// TwinCAT 3 PLC project PLC_Base
// ProgramVersion: 3.1.4024.0
// libraries:
//   Tc2_Standard, * (Beckhoff Automation GmbH)
//   Tc2_System, * (Beckhoff Automation GmbH)
//   Tc2_Utilities, * (Beckhoff Automation GmbH)
//   Tc3_Module, * (Beckhoff Automation GmbH)
// project tree:
//   DateAndTime/ FB_DateAndTimeHandling.TcPOU
//   EventLogging/ FB_EventLogger.TcPOU, FUN_EventTrigger.TcPOU
//   / MAIN.TcPOU, PlcTask.TcTTO
//   PersistantData/ PersistantDataHandling.TcPOU
//   PID/ FB_PI_Regulator.TcPOU, PRG_PI_Regulator_ProgramExample.TcPOU
//   Sequence Control/ FB_SequenceControl.TcPOU
// real-time tasks:
//   TASK PlcTask: cycle T#10ms, priority 20, ADS port 350
//   TASK PlcTask1: cycle T#10ms, priority 21, ADS port 351
//   TASK PlcTask2: cycle T#10ms, priority 22, ADS port 352
//   TASK PlcTask3: cycle T#10ms, priority 23, ADS port 353
// I/O:
//   DEVICE EtherCAT Master (Beckhoff), AmsNetId 10.75.2.8.2.1
//     EtherCAT Bus Coupler (EK1100) [EK1100 EtherCAT Coupler (2A E-Bus)]
//       ELM_Drive (ELM7211-9018) [ELM7211-9018 1Ch. Servo Terminal (48 V, 4,5 A RMS, OCT, STO, Safe Motion, TwinSAFE Logic)]
//         modules: Module 1 (SAFETY)
//       SafetyMaster 1 (EL1918) [EL1918, 8Ch. Safety Input 24V, TwinSAFE]
//         modules: Module 2 (FSLOGIC)
//       SafetyMaster 2 (EL1918) [EL1918, 8Ch. Safety Input 24V, TwinSAFE]
//         modules: Module 2 (FSLOGIC)
//     AX5000 (AX5206-0000-0215) [AX5206-0000-0215 EtherCAT Drive (SoE, 2 Ch.)]
//     AX8000(AX8620-0000-0105) [AX8620-0000-0105]
//       AX8000 Axis (AX8128-0220-0107) [AX8128-0220-0107 (1Ch. 28A servo axis, safe-motion, multi-FB) {v01.07_20240826.1_main_0107_AX8000_Axis_Daily}]
//         modules: Device, Device, Device, Device, Device, Device, Device, Device, Device, Device, Device (Safety), Device, Device, Device, Device, Device, Device, Device, Device, Device, Device, Device, Device, Device, Device, Device, Device, Device, Device, Device, Device, Ch A, Ch A, Ch A, Ch A, Ch A, Ch A, Ch A, Ch A, Ch A, Ch A, Ch A, Ch A, Ch A, Ch A, Ch A, Ch A, Ch A, Ch A, Ch A, Ch A, Ch A, Ch A, Ch A, Ch A, Ch A
//   DEVICE EtherCAT Master (NORDGear), AmsNetId 30.11.11.164.3.1
//     EtherCAT Slave To Insert In IO (NORDACpro) [NORDACpro]
//       modules: Module 1 (SK550P)
//   DEVICE Profinet Master (Siemens), AmsNetId 30.11.11.164.4.1
//     sinamics-g120c-pn [Siemens AG IO device SINAMICS G120C PN V4.7 with PROFINET-IO interface (RT, IRT and non-cyclic communications, PROFIsafe, Shared Device) 6SL3 210-1KExx-xxFx]
//       modules: Term 1 (DAP Module), Term 2 (Drive)
// variable links:
//   PLC_NORDGear/PLC_NORDGear Instance <-> EtherCAT Master (NORDGear)/EtherCAT Slave To Insert In IO (NORDACpro)
//     PlcTask Inputs/PRG_550P_ProgramExample.FRQ.HWin_ActualValue <-> Module 1 (SK550P)/Process data in/Actual value 1
//     PlcTask Inputs/PRG_550P_ProgramExample.FRQ.HWin_ActualValue @bit {16..64 step 16} <-> Module 1 (SK550P)/Process data in/Actual value {2..5}  (4 links)
//     PlcTask Inputs/PRG_550P_ProgramExample.FRQ.HWin_StatusWord <-> Module 1 (SK550P)/Process data in/Status word
//     PlcTask Outputs/PRG_550P_ProgramExample.FRQ.HWout_SetValue <-> Module 1 (SK550P)/Process data out/Set Value 1
//     PlcTask Outputs/PRG_550P_ProgramExample.FRQ.HWout_SetValue @bit {16..64 step 16} <-> Module 1 (SK550P)/Process data out/Set Value {2..5}  (4 links)
//     PlcTask Outputs/PRG_550P_ProgramExample.FRQ.HWout_StatusWord <-> Module 1 (SK550P)/Process data out/Control Word
//   PLC_Siemens/PLC_Siemens Instance <-> Profinet Master (Siemens)/sinamics-g120c-pn
//     PlcTask Inputs/PRG_G120C_ProgramExample.FRQ.HWin_Word <-> API/Term 2 (Drive)/Subterm 6 (Free telegram, PZD-6/6)/Inputs/Status word or actual value[0]
//     PlcTask Inputs/PRG_G120C_ProgramExample.FRQ.HWin_Word @bit {16..80 step 16} <-> API/Term 2 (Drive)/Subterm 6 (Free telegram, PZD-6/6)/Inputs/Status word or actual value[{1..5}]  (5 links)
//     PlcTask Outputs/PRG_G120C_ProgramExample.FRQ.Hwout_Word <-> API/Term 2 (Drive)/Subterm 6 (Free telegram, PZD-6/6)/Outputs/Control word or setpoint[0]
//     PlcTask Outputs/PRG_G120C_ProgramExample.FRQ.Hwout_Word @bit 16 <-> API/Term 2 (Drive)/Subterm 6 (Free telegram, PZD-6/6)/Outputs/Control word or setpoint[1]
//     PlcTask Outputs/PRG_G120C_ProgramExample.FRQ.Hwout_Word @bit 32 <-> API/Term 2 (Drive)/Subterm 6 (Free telegram, PZD-6/6)/Outputs/Control word or setpoint[2]
//     PlcTask Outputs/PRG_G120C_ProgramExample.FRQ.Hwout_Word @bit 48 <-> API/Term 2 (Drive)/Subterm 6 (Free telegram, PZD-6/6)/Outputs/Control word or setpoint[3]

CONFIGURATION PLC_Base
    RESOURCE PLC ON TwinCAT3
        TASK PlcTask(INTERVAL := T#10ms, PRIORITY := 23);
        PROGRAM MAIN WITH PlcTask : MAIN;
    END_RESOURCE
END_CONFIGURATION

// ---- MAIN.TcPOU
PROGRAM MAIN
VAR
END_VAR

PRG_PI_Regulator_ProgramExample();

END_PROGRAM

// ---- PID/PRG_PI_Regulator_ProgramExample.TcPOU
PROGRAM PRG_PI_Regulator_ProgramExample
VAR
	PID_Instance :				FB_PI_Regulator;
	Out_Error :					LREAL;
	Out_LoopOutput :			LREAL;
	Out_DutyOutput :			BOOL;
	Sts_DeadBandActive :		BOOL;
	Sts_LastReactionTime :		DINT;
	Sts_LastReactionTime_Offset :		DINT;
	SP_Old :					LREAL;
	SP_ChangeTON :				TON;
	Step_SIM :					INT;
	Step_SIM_Old :					INT;
	StepTON :					TON;
	SIMDampingFactor :			LREAL :=1.0;
	SIM_OvershootSUB :			LREAL :=10.0; 
	
END_VAR

SP_ChangeTON(IN:=PID_Instance.In_SP = SP_Old , PT:=T#2S , Q=> , ET=> );
IF SP_Old <> PID_Instance.In_SP THEN
		SP_Old := PID_Instance.In_SP;
END_IF
// PID Regulator
PID_Instance(Out_Error=>Out_Error , 
	Out_LoopOutput=>Out_LoopOutput , 
	Out_DutyOutput=>Out_DutyOutput,
	Sts_DeadBandActive=>Sts_DeadBandActive ,	
    Sts_LastReactionTime=>Sts_LastReactionTime_Offset);
	
Sts_LastReactionTime := Sts_LastReactionTime_Offset - 2000;
	
// SIM Control
	StepTON(IN:=Step_SIM_Old = Step_SIM , PT:=T#16D , Q=> , ET=> );
	IF Step_SIM_Old <> Step_SIM THEN
		Step_SIM_Old := Step_SIM;
	END_IF
	
	CASE Step_SIM OF
		
		0:
			IF StepTON.ET > INT_TO_TIME(PID_Instance.In_DutyCycle) AND SP_ChangeTON.Q THEN
				PID_Instance.In_PV := PID_Instance.In_PV + ((Out_LoopOutput) * SIMDampingFactor);	
				
				Step_SIM := 10;
			END_IF
		10:
			IF StepTON.ET > T#20MS THEN
				Step_SIM := 0;
			END_IF
			
	
	
	END_CASE

END_PROGRAM

// ---- PID/FB_PI_Regulator.TcPOU
FUNCTION_BLOCK FB_PI_Regulator
VAR_INPUT
	In_SP :				LREAL;
	In_PV :				LREAL;	
	In_DutyCycle :		INT;
	Cfg_P_Gain :		LREAL;
	Cfg_I_Gain :		LREAL;
	Cfg_D_Gain :		LREAL;
	Cfg_DeadBand :		LREAL;
	Cfg_FeedForward :	LREAL;
END_VAR
VAR_OUTPUT
	Out_Error :		LREAL;
	Out_LoopOutput :	LREAL;
	Out_DutyOutput :	BOOL;
	Sts_DeadBandActive :	BOOL;
	Sts_LastReactionTime :	DINT;
END_VAR
VAR
	
	DutyCycleTON :		TON;	
	P_LoopOutput :	LREAL;
	I_LoopOutput :	LREAL;
	
	DeadbandMin :	LREAL;
	DeadbandMax :	LREAL;
	ReactionTimeTON :	TON;
	ReactionTimeONS :	R_TRIG;
	
	Lo_DeadBandActive :	BOOL;
END_VAR

DutyCycleTON(IN:=NOT DutyCycleTON.Q , PT:=INT_TO_TIME(In_DutyCycle) , Q=> , ET=> );

// DeadBand
IF Cfg_DeadBand<> 0 THEN

IF In_PV < DeadbandMax AND In_PV > DeadbandMin THEN
	Sts_DeadBandActive :=1;
	ELSE
	Sts_DeadBandActive :=0;
END_IF

ReactionTimeONS(CLK:=Sts_DeadBandActive , Q=> );

IF ReactionTimeONS.Q THEN
	Sts_LastReactionTime := TIME_TO_DINT(ReactionTimeTON.ET);
END_IF

ReactionTimeTON(IN:= NOT Sts_DeadBandActive , PT:=T#16D , Q=> , ET=> );
ELSE
	
DeadbandMin := In_SP - 0.1;
DeadbandMax := In_SP + 0.1;	
IF In_PV < DeadbandMax AND In_PV > DeadbandMin THEN
	Lo_DeadBandActive :=1;
	ELSE
	Lo_DeadBandActive :=0;
END_IF

ReactionTimeONS(CLK:=Lo_DeadBandActive , Q=> );

IF ReactionTimeONS.Q THEN
	Sts_LastReactionTime := TIME_TO_DINT(ReactionTimeTON.ET);
END_IF

ReactionTimeTON(IN:= NOT Lo_DeadBandActive , PT:=T#16D , Q=> , ET=> );
END_IF	



//Regulation
IF DutyCycleTON.Q AND NOT Sts_DeadBandActive THEN

Out_Error := In_SP - In_PV;

// P
P_LoopOutput := Cfg_P_Gain*Out_Error;

// I
I_LoopOutput := Out_Error * Cfg_I_Gain;


// Calculate Output

Out_LoopOutput := P_LoopOutput + I_LoopOutput + Cfg_FeedForward;

END_IF

END_FUNCTION_BLOCK

// ---- DateAndTime/FB_DateAndTimeHandling.TcPOU
FUNCTION_BLOCK FB_DateAndTimeHandling
VAR_INPUT
END_VAR
VAR_OUTPUT
END_VAR
VAR
	
	
	TimeStruct :					Tc2_Utilities.TIMESTRUCT;
	fbGetTime:						NT_GetTime;
	
	GetTimeTON :					TON;	

END_VAR

METHOD Enable : BOOL
VAR_INPUT
END_VAR
fbGetTime(
	NETID:='' , 
	START:= GetTimeTON.Q, 
	TMOUT:= T#40S , 
	TIMESTR=>TimeStruct );
END_METHOD

PROPERTY GetActualDayOfMonthAsINT : INT
GET
GetActualDayOfMonthAsINT := WORD_TO_INT(TimeStruct.wDay);
END_GET
END_PROPERTY

PROPERTY GetActualHourAsINT : INT
GET
GetActualHourAsINT := WORD_TO_INT(TimeStruct.wHour);
END_GET
END_PROPERTY

PROPERTY GetActualMillisecondAsINT : INT
GET
GetActualMillisecondAsINT := WORD_TO_INT(TimeStruct.wMilliseconds);
END_GET
END_PROPERTY

PROPERTY GetActualMinuteAsINT : INT
GET
GetActualMinuteAsINT := WORD_TO_INT(TimeStruct.wMinute);
END_GET
END_PROPERTY

PROPERTY GetActualMonthAsINT : INT
GET
GetActualMonthAsINT := WORD_TO_INT(TimeStruct.wMonth);
END_GET
END_PROPERTY

PROPERTY GetActualSecondAsINT : INT
GET
GetActualSecondAsINT := WORD_TO_INT(TimeStruct.wSecond);
END_GET
END_PROPERTY

PROPERTY GetActualWeekdayAsINT : INT
GET
GetActualWeekdayAsINT := WORD_TO_INT(TimeStruct.wDayOfWeek);
END_GET
END_PROPERTY

PROPERTY GetActualYearAsINT : INT
GET
GetActualYearAsINT := WORD_TO_INT(TimeStruct.wYear);
END_GET
END_PROPERTY

PROPERTY GetDateAsSTRING : STRING
GET
VAR
	
	DateTime :						DT;
	ToUDT :							STRING;
	WithOutDT :						STRING;
	WithOutHyphen :					STRING;
	WithGap :						STRING;
	DateTimeString :				STRING;
	TimeString :					STRING;	

END_VAR
//Date To String
	//Makes TimeStruct to DateTime
	DateTime := SYSTEMTIME_TO_DT(TIMESTR:= TimeStruct);
	
	//Makes DateTime to String
	ToUDT := DT_TO_STRING(DateTime);
	
	//Delete #DT from String
	WithOutDT := Tc2_Standard.DELETE(STR:=ToUDT, LEN:=4,POS:=0);
	
	//Delete hyphen between date and time
	WithOutHyphen:=Tc2_Standard.DELETE(STR:=WithOutDT, LEN:=1,POS:=11);
	
	//Insert a gap between date and time	
	WithGap := Tc2_Standard.INSERT(STR1:=WithOutHyphen,STR2:=' ', POS:=10);
	DateTimeString := Tc2_Standard.DELETE(STR:=WithGap, LEN:=6,POS:=0);
	GetDateAsSTRING := Tc2_Standard.DELETE(STR:=DateTimeString, LEN:=7,POS:=8);
END_GET
END_PROPERTY

PROPERTY GetDateTimeAsSTRING : STRING
GET
VAR

	DateTime :						DT;
	ToUDT :							STRING;
	WithOutDT :						STRING;
	WithOutHyphen :					STRING;
	WithGap :						STRING;
	DateTimeString :				STRING;
	TimeString :					STRING;	

END_VAR
//Date To String
	//Makes TimeStruct to DateTime
	DateTime := SYSTEMTIME_TO_DT(TIMESTR:= TimeStruct);
	
	//Makes DateTime to String
	ToUDT := DT_TO_STRING(DateTime);
	
	//Delete #DT from String
	WithOutDT := Tc2_Standard.DELETE(STR:=ToUDT, LEN:=4,POS:=0);
	
	//Delete hyphen between date and time
	WithOutHyphen:=Tc2_Standard.DELETE(STR:=WithOutDT, LEN:=1,POS:=11);
	
	//Insert a gap between date and time	
	WithGap := Tc2_Standard.INSERT(STR1:=WithOutHyphen,STR2:=' ', POS:=10);
	DateTimeString := Tc2_Standard.DELETE(STR:=WithGap, LEN:=6,POS:=0);
	TimeString := Tc2_Standard.DELETE(STR:=DateTimeString, LEN:=7,POS:=0);
	GetDateTimeAsSTRING := DateTimeString;
END_GET
END_PROPERTY

PROPERTY GetRawDateTimeAsSTRING : STRING
GET
VAR
	
	DateTime :						DT;
	ToUDT :							STRING;
	WithOutDT :						STRING;
	EmptyString :					STRING(1);
	DateTimeString :				STRING;
	TimeString :					STRING;	

END_VAR
//Makes TimeStruct to DateTime
	DateTime := SYSTEMTIME_TO_DT(TIMESTR:= TimeStruct);
	
	//Makes DateTime to String
	ToUDT := DT_TO_STRING(DateTime);

	
	//Delete #DT from String
	WithOutDT := Tc2_Standard.DELETE(STR:=ToUDT, LEN:=4,POS:=0);

	//Delete hyphen between date and time
	GetRawDateTimeAsSTRING:= Tc2_Standard.REPLACE(STR1:=WithOutDT , STR2:=' ' , L:=1 , P:=11 ); //Tc2_Standard.DELETE(STR:=WithOutDT, LEN:=1,POS:=11);
END_GET
END_PROPERTY

PROPERTY GetTimeAsSTRING : STRING
GET
VAR

	DateTime :						DT;
	ToUDT :							STRING;
	WithOutDT :						STRING;
	WithOutHyphen :					STRING;
	WithGap :						STRING;
	DateTimeString :				STRING;
	TimeString :					STRING;	

END_VAR
//Date To String
	//Makes TimeStruct to DateTime
	DateTime := SYSTEMTIME_TO_DT(TIMESTR:= TimeStruct);
	
	//Makes DateTime to String
	ToUDT := DT_TO_STRING(DateTime);
	
	//Delete #DT from String
	WithOutDT := Tc2_Standard.DELETE(STR:=ToUDT, LEN:=4,POS:=0);
	
	//Delete hyphen between date and time
	WithOutHyphen:=Tc2_Standard.DELETE(STR:=WithOutDT, LEN:=1,POS:=11);
	
	//Insert a gap between date and time	
	WithGap := Tc2_Standard.INSERT(STR1:=WithOutHyphen,STR2:=' ', POS:=10);
	DateTimeString := Tc2_Standard.DELETE(STR:=WithGap, LEN:=6,POS:=0);
	GetTimeAsSTRING := Tc2_Standard.DELETE(STR:=DateTimeString, LEN:=7,POS:=0);
END_GET
END_PROPERTY

END_FUNCTION_BLOCK

// ---- EventLogging/FB_EventLogger.TcPOU
FUNCTION_BLOCK FB_EventLogger
VAR_INPUT
	ModuleName 			: STRING;
	NewMessageText 		: STRING(250);	
	ClearEventLog 		: BOOL;
	logEnableTimestamp		: BOOL;
END_VAR
VAR_OUTPUT
	LastLoggedMessage 	: STRING(250);
END_VAR
VAR_IN_OUT
	EventLogArray 		: ARRAY [1..100] OF STRING(250);
END_VAR
VAR
	NewMessage_Cpy 		: STRING(250);
	NewMessage_OLD 		: STRING(250);
	AddtoLogMessage 	: STRING(250);
	EmptyString 		: STRING:='';	
	StringFIND 			: INT;
	PrefixLength 		: INT;
	PrefixStartPlace 	: INT;
	Idx 				: INT;
	DateTimeHandeling 		: FB_DateAndTimeHandling;
	namelength 			: INT;
END_VAR

DateTimeHandeling.Enable();
IF NewMessageText <> NewMessage_OLD THEN
	NewMessage_OLD := NewMessageText;
	NewMessage_Cpy := NewMessageText;
	
	namelength := LEN(ModuleName);
	IF Namelength > 0 THEN
		IF logEnableTimestamp THEN
			AddtoLogMessage := CONCAT(DateTimeHandeling.GetDateTimeAsSTRING,' - ');
			AddtoLogMessage := CONCAT(AddtoLogMessage,ModuleName);
			AddtoLogMessage := CONCAT(AddtoLogMessage,' - ');
			AddtoLogMessage := CONCAT(AddtoLogMessage,NewMessage_Cpy);
		ELSE
			AddtoLogMessage := CONCAT(ModuleName,' - ');
			AddtoLogMessage := CONCAT(AddtoLogMessage,NewMessage_Cpy);
		END_IF	
	ELSE
		IF logEnableTimestamp THEN
			AddtoLogMessage := CONCAT(DateTimeHandeling.GetDateTimeAsSTRING,' - ');
			AddtoLogMessage := CONCAT(AddtoLogMessage,NewMessage_Cpy);
		ELSE
			AddtoLogMessage := NewMessage_Cpy;
		END_IF	
	END_IF

	FOR Idx := 100 TO 2 BY -1 DO
  			EventLogArray[Idx] := EventLogArray[Idx-1] ;
	END_FOR ;
		EventLogArray[1] :=AddtoLogMessage;
		LastLoggedMessage := AddtoLogMessage;
END_IF

IF ClearEventLog THEN
	FOR Idx := 100 TO 2 BY -1 DO
  			EventLogArray[Idx] := '' ;
	END_FOR ;
	ClearEventLog :=0;
END_IF

END_FUNCTION_BLOCK

// ---- EventLogging/FUN_EventTrigger.TcPOU
FUNCTION FUN_EventTrigger : BOOL
VAR_INPUT
	IN 					: STRING(250);
	ModuleName 			: STRING;
	MessageText 		: STRING(250);
END_VAR
VAR
	
	STRINGLENGTH :			INT;
	ModuleNameOK :			BOOL;
	MessageTypeOK :			BOOL;
	MessageTextOK :			BOOL;
END_VAR

StringLength := LEN(IN);

IF StringLength <> 0 THEN
		
			STRINGLENGTH := FIND(IN,ModuleName);
			IF STRINGLENGTH > 0 THEN
				ModuleNameOK :=1;
			END_IF
			STRINGLENGTH := FIND(IN,MessageText);
			IF STRINGLENGTH > 0 THEN
				MessageTextOK :=1;
			END_IF
			
		IF ModuleNameOK AND MessageTextOK THEN
			EventTrigger2 :=1;
		END_IF
		
END_IF

END_FUNCTION

// ---- PersistantData/PersistantDataHandling.TcPOU
FUNCTION_BLOCK PersistantDataHandling
VAR_INPUT
END_VAR
VAR_OUTPUT
END_VAR
VAR

	FB_WriteNow :				WritePersistentData;	

END_VAR

METHOD Enable : BOOL
VAR_INPUT
END_VAR
FB_WriteNow(NETID:='',PORT:=TwinCAT_SystemInfoVarList._AppInfo.AdsPort);
END_METHOD

METHOD WriteDataNow : BOOL
VAR
	WritePersistantDataSTEP : INT;
END_VAR
CASE WritePersistantDataSTEP OF
	
	0:
		FB_WriteNow.START := FALSE;
		WritePersistantDataSTEP := 2;
		
	2:
		FB_WriteNow.START := FALSE;
		WritePersistantDataSTEP := 5;
		
	5:

		FB_WriteNow.START := TRUE;
		WritePersistantDataSTEP := 10;
		IF FB_WriteNow.ERR THEN
			WritePersistantDataSTEP := 666;
			FB_WriteNow.START := FALSE;
		END_IF
		
	10:
		IF NOT FB_WriteNow.BUSY THEN
			FB_WriteNow.START := FALSE;
			IF NOT FB_WriteNow.ERR THEN
				WritePersistantDataSTEP := 20;
			ELSE
				WritePersistantDataSTEP := 666;
				FB_WriteNow.START := FALSE;
			END_IF
		END_IF
	20:
		FB_WriteNow.START := FALSE;
		WriteDataNow := TRUE;


END_CASE
END_METHOD

METHOD WriteDataWithTimeInterval : BOOL
VAR_INPUT
	
	TimeInterval :			TIME;

END_VAR
VAR
	WritePersistantDataIntervalSTEP :	INT;
	WaitTimeTON :						TON;
END_VAR
WaitTimeTON(IN:=WritePersistantDataIntervalSTEP = 30 , PT:=TimeInterval , Q=> , ET=> );

CASE WritePersistantDataIntervalSTEP OF
	
	0:
		FB_WriteNow.START := FALSE;
		WritePersistantDataIntervalSTEP := 2;
		
	2:
		FB_WriteNow.START := FALSE;
		WritePersistantDataIntervalSTEP := 5;
		
	5:
		FB_WriteNow.START := TRUE;
		WritePersistantDataIntervalSTEP := 10;
			
	10:
		IF NOT FB_WriteNow.BUSY THEN
			FB_WriteNow.START := FALSE;
			WriteDataWithTimeInterval := TRUE;
			IF NOT FB_WriteNow.ERR THEN
				WritePersistantDataIntervalSTEP := 20;
			ELSE
				WritePersistantDataIntervalSTEP := 666;
				FB_WriteNow.START := FALSE;
			END_IF
		END_IF
		
	20:
		IF TimeInterval > T#0MS THEN
			WritePersistantDataIntervalSTEP := 30;
			WriteDataWithTimeInterval := FALSE;
		END_IF
		
	30:
		IF WaitTimeTON.Q THEN
			WritePersistantDataIntervalSTEP := 0;
		END_IF
		

END_CASE
END_METHOD

END_FUNCTION_BLOCK

// ---- Sequence Control/FB_SequenceControl.TcPOU
FUNCTION_BLOCK FB_SequenceControl
VAR_INPUT
	step 					: UDINT;
	stepDescriptionText		: STRING(250);
	logEnableStepInfo		: BOOL;
	logEnableADSLogging		: BOOL;
END_VAR
VAR_OUTPUT
	stepFirstscan 			: BOOL;
	StepActiveTimer 		: TIME;
	ScanCounter 			: ULINT;
	Error					: BOOL;
	ErrorStep				: UDINT;
	LastStepInfo 			: STRING(250);
	NewMessageReady 		: BOOL;
END_VAR
VAR
	stepLast 				: UDINT;
	stepTimer 				: TON;
	LastStepDescriptionText : STRING(250);
	
	StepChangeONS 			: R_TRIG;
	
	StringLength 			: INT;
	StringERRORFind 		: INT;
	StringWARNINGFind 		: INT;
	StringINFORMATIONFind 	: INT;
	Idx 					: INT;
	NewStringTEMP 			: STRING(250);
	NewStringTEMP_Old		: STRING(250);
	DateAndTimeSTRING 		: STRING;
	
	ParsedmessageSTRING		: STRING(250);
	TXTCategory				: INT;
END_VAR

stepTimer(PT := T#24D, ET =>StepActiveTimer);

IF stepLast <> Step THEN
	
	LastStepInfo := CONCAT('Step : ',UDINT_TO_STRING(stepLast));
	
	LastStepInfo := CONCAT(LastStepInfo,' - ');
	LastStepInfo := CONCAT(LastStepInfo,stepDescriptionText);
		
	IF logEnableStepInfo THEN
		IF TIME_TO_DINT(StepActiveTimer) > 0 THEN
			LastStepInfo := 'StepTime : ';
			LastStepInfo := CONCAT(LastStepInfo,TIME_TO_STRING(StepActiveTimer));
		END_IF
		LastStepInfo := CONCAT(LastStepInfo,', ScanCount : ');
		LastStepInfo := CONCAT(LastStepInfo,LINT_TO_STRING(ScanCounter));
	END_IF
		
	stepTimer.IN := 0;
	stepFirstscan := TRUE;
	ScanCounter :=0;
	stepLast := step;
	Error :=0;
	ErrorStep :=0;
	LogNow();
ELSE
	stepFirstscan := FALSE;
	stepTimer.IN := 1;
	NewMessageReady := FALSE;
END_IF

// Timer
ScanCounter := ScanCounter +1;

ACTION LogNow:
NewStringTEMP :='';
StringLength := LEN(stepDescriptionText);						
	IF logEnableADSLogging THEN
		IF StringLength <> 0 THEN
				
			STRINGLENGTH := FIND(stepDescriptionText,'STATUS');
			IF STRINGLENGTH <> 0 THEN
				stepDescriptionText := DELETE(STR:=stepDescriptionText, LEN:=7,POS:=1);
				IF logEnableStepInfo THEN
					stepDescriptionText := CONCAT(stepDescriptionText,' - ');
					stepDescriptionText := CONCAT(stepDescriptionText,LastStepInfo);
				END_IF
				ADSLOGSTR(msgCtrlMask:=ADSLOG_MSGTYPE_LOG , msgFmtStr:=stepDescriptionText , strArg:='' );
			ELSIF STRINGLENGTH <> 0 THEN
		
			STRINGLENGTH := FIND(stepDescriptionText,'ERROR');
				ErrorStep := Step;
				Error := 1;
				stepDescriptionText := DELETE(STR:=stepDescriptionText, LEN:=6,POS:=1);
				IF logEnableStepInfo THEN
					stepDescriptionText := CONCAT(stepDescriptionText,' - ');
					stepDescriptionText := CONCAT(stepDescriptionText,LastStepInfo);
				END_IF
				ADSLOGSTR(msgCtrlMask:=ADSLOG_MSGTYPE_ERROR , msgFmtStr:=ParsedmessageSTRING , strArg:='' );
			ELSIF STRINGLENGTH <> 0 THEN
			
			STRINGLENGTH := FIND(stepDescriptionText,'WARNING');

				stepDescriptionText := DELETE(STR:=stepDescriptionText, LEN:=8,POS:=1);
				IF logEnableStepInfo THEN
					stepDescriptionText := CONCAT(stepDescriptionText,' - ');
					stepDescriptionText := CONCAT(stepDescriptionText,LastStepInfo);
				END_IF
				ADSLOGSTR(msgCtrlMask:=ADSLOG_MSGTYPE_WARN , msgFmtStr:=ParsedmessageSTRING , strArg:='' );
			ELSIF STRINGLENGTH <> 0 THEN

			STRINGLENGTH := FIND(stepDescriptionText,'INFORMATION');

				stepDescriptionText := DELETE(STR:=stepDescriptionText, LEN:=12,POS:=1);
				IF logEnableStepInfo THEN
					stepDescriptionText := CONCAT(stepDescriptionText,' - ');
					stepDescriptionText := CONCAT(stepDescriptionText,LastStepInfo);
				END_IF
				ADSLOGSTR(msgCtrlMask:=ADSLOG_MSGTYPE_LOG , msgFmtStr:=stepDescriptionText , strArg:='' );
			ELSE
				IF logEnableStepInfo THEN
					stepDescriptionText := CONCAT(stepDescriptionText,' - ');
					stepDescriptionText := CONCAT(stepDescriptionText,LastStepInfo);
				END_IF
				ADSLOGSTR(msgCtrlMask:=ADSLOG_MSGTYPE_LOG , msgFmtStr:=stepDescriptionText , strArg:='' );
			END_IF
		END_IF
							
		
	END_IF
	
	IF LastStepDescriptionText <> stepDescriptionText THEN
		NewMessageReady := TRUE;
		LastStepDescriptionText := stepDescriptionText;
	END_IF
END_ACTION

END_FUNCTION_BLOCK
